// TIA Portal project "WordClock_V17" (V17)

(* hardware
DEVICE "S7-1200-Station_1"  S7-1200 Station
   slot 0: "Baugruppenträger_0"  Rack  V1.0
   slot 1: "PLC"  CPU 1214C DC/DC/DC  6ES7 214-1AG40-0XB0  V4.1
   slot 3: "AQ 1x12BIT_1"  6ES7 232-4HA30-0XB0  V1.0
*)

// ===== PLC "PLC"  CPU 1214C DC/DC/DC =====

VAR_GLOBAL   // PLC tag table "Standard-Variablentabelle"
   "System_Byte" AT %MB100 : Byte;
   "FirstScan" AT %M100.0 : Bool;
   "DiagStatusUpdate" AT %M100.1 : Bool;
   "AlwaysTRUE" AT %M100.2 : Bool;
   "AlwaysFALSE" AT %M100.3 : Bool;
   "Clock_Byte" AT %MB110 : Byte;
   "Clock_10Hz" AT %M110.0 : Bool;
   "Clock_5Hz" AT %M110.1 : Bool;
   "Clock_2.5Hz" AT %M110.2 : Bool;
   "Clock_2Hz" AT %M110.3 : Bool;
   "Clock_1.25Hz" AT %M110.4 : Bool;
   "Clock_1Hz" AT %M110.5 : Bool;
   "Clock_0.625Hz" AT %M110.6 : Bool;
   "Clock_0.5Hz" AT %M110.7 : Bool;
END_VAR

DATA_BLOCK "VersionInput"   // DB1
{ S7_Optimized_Access := 'FALSE' }
VERSION : 0.1
   VAR
      AutoTest : Bool;
      "Version" : String := 'WorkClock V2.0';
   END_VAR
BEGIN
END_DATA_BLOCK

DATA_BLOCK "DigInput"   // DB2
{ S7_Optimized_Access := 'FALSE' }
VERSION : 0.1
   VAR
      DateTime : DTL;   // Datum / Zeit
   END_VAR
BEGIN
END_DATA_BLOCK

DATA_BLOCK "DigOutput"   // DB3
{ S7_Optimized_Access := 'FALSE' }
VERSION : 0.1
   VAR
      ES : Bool;
      IST : Bool;
      BALD : Bool;
      GLEICH : Bool;
      VIERTEL : Bool;
      ZWANZIG : Bool;
      ZEHN_MINUTEN : Bool;
      FÜNF_MINUTEN : Bool;
      VOR : Bool;
      NACH : Bool;
      HALB : Bool;
      ZWÖLF : Bool;
      ELF : Bool;
      ZEHN_STUNDEN : Bool;
      NEUN : Bool;
      ACHT : Bool;
      SIEBEN : Bool;
      SECHTS : Bool;
      FÜNF_STUNDEN : Bool;
      VIER : Bool;
      DREI : Bool;
      ZWEI : Bool;
      EINS : Bool;
      UHR : Bool;
   END_VAR
BEGIN
END_DATA_BLOCK

DATA_BLOCK "AnInput"   // DB4
{ S7_Optimized_Access := 'FALSE' }
VERSION : 0.1
BEGIN
END_DATA_BLOCK

DATA_BLOCK "AnOutput"   // DB5
{ S7_Optimized_Access := 'FALSE' }
VERSION : 0.1
BEGIN
END_DATA_BLOCK

DATA_BLOCK "DeleteMe_DB"   // DB6
{ S7_Optimized_Access := 'TRUE' }
VERSION : 0.1
// stored: InstanceOfName DeleteMe
"DeleteMe"
BEGIN
END_DATA_BLOCK

FUNCTION_BLOCK "DeleteMe"   // FB1, SCL
{ S7_Optimized_Access := 'TRUE' }
VERSION : 0.1
   VAR
      Bitmuster : Array[0..256] of Int;
      Init : Bool;
      Zeiger : Int;
      Ergebnis : Word;
      Ascii : Word;
   END_VAR
   VAR CONSTANT
      P1R : Int := 2#0000_0000_0001;
      P1L : Int := 2#0000_0000_0010;
      P2R : Int := 2#0000_0000_0100;
      P2L : Int := 2#0000_0000_1000;
      P3R : Int := 2#0000_0001_0000;
      P3L : Int := 2#0000_0010_0000;
      P4R : Int := 2#0000_0100_0000;
      P4L : Int := 2#0000_1000_0000;
      P5R : Int := 2#0001_0000_0000;
      P5L : Int := 2#0010_0000_0000;
   END_VAR
BEGIN

   IF NOT #Init THEN
       FOR #Zeiger := 0 TO 255 DO
           #Bitmuster[#Zeiger] := 0;
       END_FOR;

       #Bitmuster[16#41] := #P1R + #P5L; //65 A
       #Bitmuster[16#42] := #P1R + #P4L; //66 B
       #Bitmuster[16#44] := #P2R + #P5L; //68 D
       #Bitmuster[16#45] := #P1R + #P3L; //69 E
       #Bitmuster[16#46] := #P2R + #P4L; //70 F
       #Bitmuster[16#47] := #P3R + #P5L; //71 G
       #Bitmuster[16#48] := #P1R + #P2L; //72 H
       #Bitmuster[16#49] := #P2R + #P3L; //73 I
       #Bitmuster[16#4B] := #P3R + #P4L; //75 K
       #Bitmuster[16#4C] := #P4R + #P5L; //76 L

       #Bitmuster[16#4D] := #P1L + #P2R; //77 M
       #Bitmuster[16#4E] := #P2L + #P3R; //78 N
       #Bitmuster[16#4F] := #P3L + #P4R; //79 O
       #Bitmuster[16#50] := #P4L + #P5R; //80 P
       #Bitmuster[16#52] := #P1L + #P3R; //82 R
       #Bitmuster[16#53] := #P2L + #P4R; //83 S
       #Bitmuster[16#54] := #P3L + #P5R; //84 T
       #Bitmuster[16#56] := #P1L + #P4R; //86 V
       #Bitmuster[16#57] := #P2L + #P5R; //87 W
       #Bitmuster[16#59] := #P1L + #P5R; //89 Y    
   END_IF;

   #Ascii := "DigInput".S1;
   #Ergebnis := #Bitmuster[#Ascii];

   POKE(area := 16#84,
        dbNumber := 3,
        byteOffset := 0,
        value := #Ergebnis.%B0);
   POKE(area := 16#84,
        dbNumber := 3,
        byteOffset := 1,
        value := #Ergebnis.%B1);
END_FUNCTION_BLOCK

FUNCTION "DatenRangieren" : Void   // FC1, SCL
{ S7_Optimized_Access := 'TRUE' }
VERSION : 0.1
   VAR_TEMP
      ErstesByte : Byte;
      ZweitesByte : Byte;
   END_VAR
BEGIN
   IF "VersionInput".AutoTest THEN
       ; //  Es werden nur die Datenbausteine verwendet  
   ELSE
       // Digitale Eingänge I0.0 - I1.7 in den Datenbaustein DigInput DB2 kopieren
       // IB0 --> DB2 Byte 0
       // IB1 --> DB2 Byte 1
       // Area 16#81 --> Input
       // Area 16#82 --> Output
       // Area 16#84 --> DB
       #ErstesByte := PEEK(area := 16#81, dbNumber := 0, byteOffset := 0);
       #ZweitesByte := PEEK(area := 16#81, dbNumber := 0, byteOffset := 1);

       POKE(area := 16#84,
            dbNumber := 2,
            byteOffset := 0,
            value := #ErstesByte);
       POKE(area := 16#84,
            dbNumber := 2,
            byteOffset := 1,
            value := #ZweitesByte);

       // DB DigOutput auf die Ausgänge Q0.0 - Q1.7 kopieren
       // DB3 Byte 0 --> QB0
       // DB3 Byte 1 --> QB1
       #ErstesByte := PEEK(area := 16#84, dbNumber := 3, byteOffset := 0);
       #ZweitesByte := PEEK(area := 16#84, dbNumber := 3, byteOffset := 1);

       POKE(area := 16#82,
            dbNumber := 0,
            byteOffset := 0,
            value := #ErstesByte);
       POKE(area := 16#82,
            dbNumber := 0,
            byteOffset := 1,
            value := #ZweitesByte);
   END_IF;
END_FUNCTION

ORGANIZATION_BLOCK "Main"   // OB1, LAD, ProgramCycle
TITLE = "Main Program Sweep (Cycle)"
{ S7_Optimized_Access := 'TRUE' }
VERSION : 0.1
   VAR_INPUT
      Initial_Call : Bool;   // Initial call of this OB
      Remanence : Bool;   // =True, if remanent data are available
   END_VAR
BEGIN

REGION Network 1: -Q1
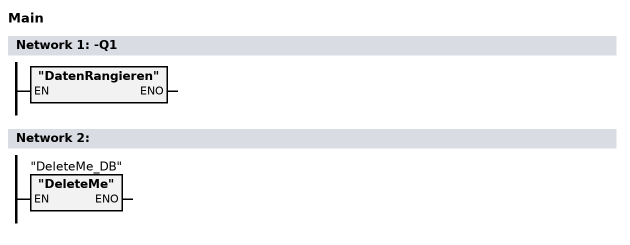
   RUNG wire#powerrail
      "DatenRangieren"()
   END_RUNG
   // the same network as SCL:
   "DatenRangieren"();
END_REGION

REGION Network 2
   RUNG wire#powerrail
      "DeleteMe_DB"()
   END_RUNG
   // the same network as SCL:
   "DeleteMe_DB"();   // "DeleteMe"
END_REGION
END_ORGANIZATION_BLOCK

ORGANIZATION_BLOCK "Startup"   // OB100, SCL, Startup
TITLE = "Complete Restart"
{ S7_Optimized_Access := 'TRUE' }
VERSION : 0.1
   VAR_INPUT
      LostRetentive : Bool;   // True if retentive data are lost
      LostRTC : Bool;   // True if date and time are lost
   END_VAR
BEGIN
   "VersionInput".AutoTest := TRUE;

   POKE(area := 16#84,     // DB
        dbNumber := 3,     // DigOutput
        byteOffset := 0,   // Byte 0
        value := byte#0);  // löschen

   POKE(area := 16#84,     // DB
        dbNumber := 3,     // Digoutput
        byteOffset := 1,   // Byte 1
        value := byte#0);  // löschen
END_ORGANIZATION_BLOCK